(* PLC project Counter (OSIE), Unknown Unnamed 1 *)
(* stored: creationDateTime 2021-05-14T14:33:11, modificationDateTime 2022-01-18T16:31:25 *)

FUNCTION_BLOCK CounterST
  VAR_OUTPUT
    Out0 : INT;
  END_VAR
  VAR
    Cnt0 : INT;
  END_VAR
  VAR_EXTERNAL
    Coupler0_Relay0 : DINT;
    Coupler0_Relay1 : DINT;
    Coupler0_Relay2 : DINT;
    Coupler0_Relay3 : DINT;
    Coupler1_Relay0 : DINT;
    Coupler1_Relay1 : DINT;
    Coupler1_Relay2 : DINT;
    Coupler1_Relay3 : DINT;
  END_VAR

            Cnt0 := Cnt0 + 1;
IF Cnt0 = 100 THEN
    Coupler0_Relay0 := Coupler0_Relay0 + 1;
    Coupler1_Relay0 := Coupler0_Relay0;
    Cnt0 := 0;
END_IF;
Out0 := Cnt0;
          
END_FUNCTION_BLOCK

PROGRAM plc_prg
  VAR
    CounterST0 : CounterST;
  END_VAR

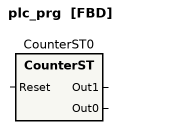
(* FBD diagram, written out as Structured Text *)
(* This PLC program is used in automated testing of beremiz' runtime / coupler integration *)
CounterST0();
END_PROGRAM

CONFIGURATION config
  VAR_GLOBAL
    Coupler0_Relay0 AT %QD1.0 : DINT := 0;  (* OPC-UA relay 0 at coupler 0 *)
    Coupler0_Relay1 AT %QD1.1 : DINT := 0;  (* OPC-UA relay 1 at coupler 0 *)
    Coupler0_Relay2 AT %QD1.2 : DINT := 0;  (* OPC-UA relay 2 at coupler 0 *)
    Coupler0_Relay3 AT %QD1.3 : DINT := 0;  (* OPC-UA relay 3 at coupler 0 *)
    Coupler1_Relay0 AT %QD0.0 : DINT := 0;  (* OPC-UA relay 0 at coupler 1 *)
    Coupler1_Relay1 AT %QD0.1 : DINT := 0;  (* OPC-UA relay 1 at coupler 1 *)
    Coupler1_Relay2 AT %QD0.2 : DINT := 0;  (* OPC-UA relay 2 at coupler 1 *)
    Coupler1_Relay3 AT %QD0.3 : DINT := 0;  (* OPC-UA relay 3 at coupler 1 *)
  END_VAR
  RESOURCE resource1 ON PLC
    TASK task0(INTERVAL := T#20ms, PRIORITY := 0);
    PROGRAM instance0 WITH task0 : plc_prg;
  END_RESOURCE
END_CONFIGURATION
